PROGRAM MAIN
VAR
END_VAR

Main_Algorithm();

END_PROGRAM

(* stored: Version 1.1.0.1, ProductVersion 3.1.4026.11
   POU MAIN: Id {314d22f9-fd1b-4489-86ae-4464ca2439f5}, SpecialFunc None *)
